PROGRAM MAIN
VAR
    bButton : BOOL;   // Buton (giris) - simdilik sanal
    bLED    : BOOL;   // LED (cikis)  - simdilik sanal
END_VAR

bLED := bButton;

END_PROGRAM

(* stored: Version 1.1.0.1
   POU MAIN: Id {754979d4-a78e-4fca-8575-fe56d25142c0}, SpecialFunc None *)
